FUNCTION_BLOCK FINAL TcoAdsLogger EXTENDS TcoLogger
VAR_INPUT
END_VAR
VAR_OUTPUT
END_VAR
VAR
END_VAR

(*~
		<docu>
			<summary>
				Creates message of given category for this logger.				 
			</summary>				
		</docu>
~*)
METHOD PROTECTED  Post 
VAR_INPUT
	(*~
		<docu>
			<summary>
				Arbitrary message string.			 
			</summary>			
		</docu>
	~*)
	Message : STRING(255);
	(*~
		<docu>
			<summary>
				Message category.			 
			</summary>			
		</docu>
	~*)
	Category : eMessageCategory;	
END_VAR
// ADSLOGSTR();
END_METHOD

END_FUNCTION_BLOCK

(* stored: Version 1.1.0.1, ProductVersion 3.1.4024.9
   POU TcoAdsLogger: Id {e5b4a06d-470b-0208-1ce9-651927148720}, SpecialFunc None
   Method Post: Id {ec283f9c-2f37-0153-0dd6-cd974ad1e2f9} *)
